FUNCTION_BLOCK StartMotorsProgramAndMovementsTask EXTENDS TcoUrRoboticsTask
VAR_INPUT
	refStartMotorsAndProgramTask: REFERENCE TO StartMotorsAndProgramTask;
END_VAR 
VAR
     _moveParams:TcoAbstractions.TcoRoboticsMovementsParams;
	 
	 
END_VAR
VAR
	_startMotorsAndProgramTask: REFERENCE TO StartMotorsAndProgramTask;
END_VAR

IF NOT __ISVALIDREF(refStartMotorsAndProgramTask)  THEN
    Messenger.Post('<#Invalid reference StartMotorAndProgramTask#>', TcoCore.eMessageCategory.ProgrammingError);
    RETURN;
END_IF
_startMotorsAndProgramTask REF= refStartMotorsAndProgramTask;

IF Execute() THEN
	IF _progress = 0 THEN
		IF NOT __ISVALIDREF(inoControl) THEN
			_varInfo :=__VARINFO(inoControl);
			Messenger.Programming(_sb.Clear().Append('<#Invalid reference: #>').Append(_varInfo.Symbol).ToString()).Pin();
		ELSIF NOT __ISVALIDREF(inoConfig) THEN                                                  
			_varInfo :=__VARINFO(inoConfig);                                                    
			Messenger.Programming(_sb.Clear().Append('<#Invalid reference: #>').Append(_varInfo.Symbol).ToString()).Pin();
		ELSIF NOT __ISVALIDREF(inoStatus) THEN                                                  
			_varInfo :=__VARINFO(inoStatus);                                                    
			Messenger.Programming(_sb.Clear().Append('<#Invalid reference: #>').Append(_varInfo.Symbol).ToString()).Pin();
			ELSE
			_progress := _progress + 1;
		END_IF

	END_IF
	
	IF _progress = 1 THEN
		IF _startMotorsAndProgramTask.Invoke().Done THEN
			_progress := _progress + 1;
		END_IF

	END_IF;
	
	
	IF _progress = 2 THEN
		inoControl.GlobalSpeed := _moveParams.GlobalSpeed;
		inoControl.ToolNo := _moveParams.ToolNo;
		inoControl.WorkobjectNo := _moveParams.WorkobjectNo;
		inoControl.PointNo := _moveParams.PointNo;
		inoControl.UserSpecSpeed1 := _moveParams.UserSpecSpeed1;
		inoControl.UserSpecSpeed2 := _moveParams.UserSpecSpeed2;
		inoControl.Coordinates := _moveParams.Coordinates; 		
	
		inoControl.ActionNo := 254;
		IF inoControl.ActionNo = inoStatus.State.ActionNo THEN
			inoControl.ActionNo := 255;
			_progress:=_progress + 1;
		END_IF
	END_IF;	
	IF _progress = 3 THEN
		IF 	inoStatus.State.GlobalSpeed = _moveParams.GlobalSpeed AND
			inoStatus.State.ToolNo = _moveParams.ToolNo AND
			inoStatus.State.WorkobjectNo = _moveParams.WorkobjectNo AND
			inoStatus.State.PointNo = _moveParams.PointNo AND
			inoStatus.State.UserSpecSpeed1 = _moveParams.UserSpecSpeed1 AND
			inoStatus.State.UserSpecSpeed2 =_moveParams.UserSpecSpeed2 AND
			TcoAbstractions.CoordinatesAreEqual(inoStatus.State.Coordinates,_moveParams.Coordinates,0.01,0.01,0.01,0.01,0.01,0.01) THEN
			inoControl.ActionNo := 255;
			_progress:=_progress + 1;
		END_IF
	END_IF;	
	
	IF _progress = 4 THEN
		IF inoControl.ActionNo = inoStatus.State.ActionNo THEN
			_progress:=_progress + 1;
		END_IF
	END_IF;	
	
	
	IF _progress = 5 THEN
	
		Messenger.Info(CONCAT('<#Moving to position ID#>: ', INT_TO_STRING(_moveParams.ActionNo)));
		inoControl.ActionNo := _moveParams.ActionNo;
		IF inoControl.ActionNo = inoStatus.State.ActionNo THEN
			inoControl.ActionNo :=255;
				_progress := _progress + 1;
		END_IF
	END_IF;		
			
	IF _progress = 6 THEN
		IF inoControl.ActionNo = inoStatus.State.ActionNo THEN
			 DoneWhen(TRUE);
		END_IF
	END_IF;		

   CallTimers(TRUE);
	
	THIS^.ThrowWhen(_errorTimer.Q );
END_IF

IF  THIS^.Error AND NOT _errorMessage.Pinned THEN
	THIS^.Restore();
END_IF

METHOD PUBLIC FB_init : BOOL
VAR_INPUT
    bInitRetains : BOOL; // if TRUE, the retain variables are initialized (warm start / cold start)
    bInCopyCode : BOOL; // if TRUE, the instance afterwards gets moved into the copy code (online change)
  	ParentObject : ITcoObject;	
END_VAR
END_METHOD

METHOD INTERNAL InvokeWithParams : ITcoTaskStatus
VAR_INPUT
    inMoveParams:TcoAbstractions.TcoRoboticsMovementsParams;
END_VAR
_moveParams:=inMoveParams;
InvokeWithParams := THIS^.Invoke();
END_METHOD

(*~
	<docu>
		<summary>
			Executes when task is aborted.
		</summary>			
	</docu>	
~*)
METHOD PROTECTED OnAbort
IF  __ISVALIDREF(inoStatus) THEN   THIS^.inoStatus.ActionDescription := '<#Start motors, program and movements was aborted, while not yet completed!#>';END_IF; 
inoControl.Pause := TRUE;
END_METHOD

(*~
	<docu>
		<summary>
			Executes when task reaches the ```Done``` state .
		</summary>			
	</docu>	
~*)
METHOD PROTECTED OnDone
IF  __ISVALIDREF(inoStatus) THEN   THIS^.inoStatus.ActionDescription := '<#Start motors, program and movements finished successfully.#>'; END_IF;
_progress:=0;
END_METHOD

(*~
	<docu>
		<summary>
			Executes when task reaches the ```Error``` state.
		</summary>			
	</docu>	
~*)
METHOD PROTECTED OnError
VAR
	description: STRING;
END_VAR
description := '<#Start motors, program and movements finished with error.#>';
IF  __ISVALIDREF(inoStatus) THEN   THIS^.inoStatus.ActionDescription := description; END_IF;
THIS^._errorMessage.Error(_sb.Clear().Append(description).Append(' To restore acknowledge this alarm.').ToString()).Pin();
END_METHOD

METHOD PROTECTED OnStart
IF  __ISVALIDREF(inoStatus) THEN   THIS^.inoStatus.ActionDescription := '<#Start motors, program and movements stared.#>'; END_IF;
CallTimers(FALSE);
inoControl.Pause := TRUE;
END_METHOD

(*~
	<docu>
		<summary>
			Restores this instance to the Ready state. Can be called explicitly or from within one of the restore mechanisms.
			<para>
				See also <see cref="PlcDocu.TcoCore.TcoTask.AutoRestorable()"/>
			</para>
		</summary>			
	</docu>	
~*)
METHOD Restore : ITcoRestorable
SUPER^.Restore();
END_METHOD

END_FUNCTION_BLOCK

(* stored: Version 1.1.0.1, ProductVersion 3.1.4024.12
   POU StartMotorsProgramAndMovementsTask: Id {f028f537-40ff-0e39-1b5f-bc29bf8fda3b}, SpecialFunc None
   Method FB_init: Id {1f636cc9-df38-0f41-2996-a02bb0bc32e4}
   Method InvokeWithParams: Id {133c4759-2021-0877-2f15-0f7839f948b2}
   Method OnAbort: Id {73ba5e6d-5b1a-0ba5-1112-2acf7d78bb93}
   Method OnDone: Id {961d2822-a37e-05e0-017a-d5a83801feac}
   Method OnError: Id {ce1ed95b-5eb7-0e5c-15aa-5df39dab405a}
   Method OnStart: Id {800d6d3a-b2eb-05fa-153b-a3f836ae1839}
   Method Restore: Id {4dd95404-c425-0926-274e-50245de5593a} *)
